FUNCTION_BLOCK EMB_RES
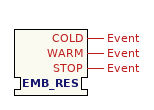
  EVENT_OUTPUT
    COLD;
    WARM;
    STOP;
  END_EVENT
END_FUNCTION_BLOCK
